FUNCTION_BLOCK FB_FSM
VAR_INPUT
	stIn		:	ST_FSM_In;
	stCtrl		:	ST_FSM_Ctrl;
	stCmd		:	ST_FSM_Cmd;
	stParams	:	ST_FSM_Params;
END_VAR
VAR_IN_OUT
	stStatus	:	ST_FSM_Status;	
END_VAR
VAR_OUTPUT	
	eStep		:	E_FSM_Step;
	tStepTime	:	TIME;
	eErrStep	:	E_FSM_Step;
	nErrId		:	DINT;
	// Digital Outputs
	stOut		:	ST_FSM_Out;	
	
END_VAR
VAR
	// FSM internal variables
	bInitialized	:	BOOL;
	eNewstep		:	E_FSM_Step;
	bEntryact		:	BOOL;
	fbTonStep		:	TON;

	(* filters on other input from plant *)
	
	(* stop request *)	
	bStopRequest	:	BOOL;
	
	// all zones are stopped
	bAllZoneStopped	:	BOOL;	
END_VAR

IF NOT bInitialized THEN
	(* here you can wait events from other controllers *)
	eNewStep := E_FSM_Step.NoStep;
	stStatus.eStep := E_FSM_Step.NeOrError;
	bEntryact := FALSE;
	bInitialized := TRUE;
ELSE
	// --- FSM Cyclical Code ----------------------------------------------
	
	// update of the enabling conditions (bStop, alarms, etc.)
	
	
	// 1. FSM Preamble ----------------------------------------------------
    // 1.a State machine disabled or failure
	IF NOT stCtrl.bEnable OR stStatus.bFailure THEN
		eNewStep := E_FSM_Step.NeOrError;
	END_IF

	// 1.b Update eStep with the required step to perform
	//     and set bEntryact to FALSE in order to enable the Entry action
	IF eNewstep <> E_FSM_Step.NoStep THEN
		stStatus.eStep := eNewstep;
		eNewstep := E_FSM_Step.NoStep;
		bEntryact := FALSE;
	END_IF;	
	
	// 1.c Do filters on signals	

	// Do requests, for example to stop the machine
	IF stCmd.bStop THEN
		bStopRequest := TRUE;
	END_IF

	// 2. The main switch-case ---------------------------------------------------
	CASE stStatus.eStep OF
    E_FSM_Step.NeOrError :
			// on entry action
			IF NOT bEntryact THEN
				stStatus.bFailure := TRUE;
				bEntryact := TRUE;
			END_IF
			
			// body
			stOut.bFixedGreen := TRUE;
			stOut.bBlinkingGreen := FALSE;
			stOut.bFixedRed := FALSE;
			stOut.bBlinkingRed := TRUE;
			stOut.bFixedYellow := FALSE;
			stOut.bBlinkingYellow := FALSE;				
			
			// next state transition
			IF stCtrl.bEnable THEN
				IF stCmd.bAck THEN
					eNewStep := E_FSM_Step.Recovering;
				END_IF
			END_IF
		
			// on exit action
			IF eNewStep <> E_FSM_Step.NoStep THEN
				nErrId := 0;
				eErrStep := E_FSM_Step.NoStep;
			END_IF

		// Recovering ---------------------------------			
		E_FSM_Step.Recovering :
			// on entry action
			IF NOT bEntryact THEN
				bEntryact := TRUE;
			END_IF
			
			// body	
			stOut.bFixedGreen := TRUE;
			stOut.bBlinkingGreen := FALSE;
			stOut.bFixedRed := FALSE;
			stOut.bBlinkingRed := FALSE;
			stOut.bFixedYellow := FALSE;
			stOut.bBlinkingYellow := TRUE;
			
			// next state transition
			IF stCtrl.bEnable THEN
				IF FC_AllStopped(stStatus) THEN
					eNewStep := E_FSM_Step.Stopping;
				END_IF				
			END_IF
			
			// on exit action
			IF eNewStep <> E_Z3_Step.NoStep THEN
				stStatus.bFailure := FALSE;
			END_IF

		// Stopping ---------------------------------			
		E_FSM_Step.Stopping :
			// on entry action
			IF NOT bEntryact THEN
				bEntryact := TRUE;
			END_IF
			
			// body	
			stOut.bFixedGreen := FALSE;
			stOut.bBlinkingGreen := TRUE;
			stOut.bFixedRed := FALSE;
			stOut.bBlinkingRed := FALSE;
			stOut.bFixedYellow := FALSE;
			stOut.bBlinkingYellow := TRUE;
			
			// next state transition
			IF stCtrl.bEnable THEN
				IF stStatus.tStepTime > stParams.tStoppingDelay THEN
					eNewStep := E_FSM_Step.Stop;
				END_IF				
			END_IF
			
			// on exit action
			IF eNewStep <> E_Z3_Step.NoStep THEN
			   ;
			END_IF

		// Stop ---------------------------------			
		E_FSM_Step.Stop :
			// on entry action
			IF NOT bEntryact THEN
				bEntryact := TRUE;
			END_IF
			
			// body	
			stOut.bFixedGreen := FALSE;
			stOut.bBlinkingGreen := FALSE;
			stOut.bFixedRed := TRUE;
			stOut.bBlinkingRed := FALSE;
			stOut.bFixedYellow := FALSE;
			stOut.bBlinkingYellow := TRUE;
			
			// next state transition
			IF stCtrl.bEnable AND stCmd.bStart AND NOT stCmd.bStop THEN
				eNewStep := E_FSM_Step.Running;			
			END_IF
			
			// on exit action
			IF eNewStep <> E_Z3_Step.NoStep THEN
			   ;
			END_IF						

		// Running ---------------------------------			
		E_FSM_Step.Running :
			// on entry action
			IF NOT bEntryact THEN
				bEntryact := TRUE;
			END_IF
			
			// body	
			stOut.bFixedGreen := TRUE;
			stOut.bBlinkingGreen := FALSE;
			stOut.bFixedRed := FALSE;
			stOut.bBlinkingRed := FALSE;
			stOut.bFixedYellow := FALSE;
			stOut.bBlinkingYellow := FALSE;
			
			// next state transition
			IF stCtrl.bEnable AND stCmd.bStart AND NOT stCmd.bStop THEN
				eNewStep := E_FSM_Step.Running;			
			END_IF
			
			// on exit action
			IF eNewStep <> E_Z3_Step.NoStep THEN
			   ;
			END_IF	

	
	ELSE
		// this happens also if we forget to code one step 
		eNewstep := E_FSM_Step.NeOrError;
		stStatus.eErrorStep := E_FSM_Step.Unknown;
		stStatus.nErrorID := -9;
	END_CASE;
	
	// 3. FSM Epilogue ------------------------------------------------------
	
	// Elapsed time into the current step
	fbTonStep(IN := (eNewstep = E_FSM_Step.NoStep), PT := T#500H );
	stStatus.tStepTime := fbTonStep.ET;
	
END_IF

END_FUNCTION_BLOCK

(* stored: Version 1.1.0.1
   POU FB_FSM: Id {d98d3e8f-9e6f-03e2-15bd-3508773e39b6}, SpecialFunc None *)
